(* CoDeSys 2.3 export: NETVARTLGHEADER_UDP.EXP *)

(* Data type *)
TYPE NetVarTlgHeader_Udp :
STRUCT
	dwIdentity	: DWORD := TELEGRAM_IDENT; (* Kennung für Art der UDP Message BYTE 0 = '3', 1 = 'S', 2 = '-' , 3 = Nummer der Version *)
	dwID		: DWORD;
	nIndex		: INT;
	nSubIndex	: INT;
	nItems		: INT;
	nLen		: INT;
	nCounter	: INT;
	byFlags 	: BYTE; (*Bit 0: Sende Bestätigung erwünscht*)
						 (*Bit 1: Checksumme prüfen*)
						 (*Bit 2: Ungültige Checksumme*)
	byChecksum: BYTE;
END_STRUCT
END_TYPE
